TYPE STriggeredOutput :
STRUCT
	ChangeTrigger: USINT;
END_STRUCT
END_TYPE

(* stored: Version 1.1.0.1
   DUT STriggeredOutput: Id {47df0f34-6ef2-4838-a51b-d0ca70509605} *)
